// TwinCAT 3 PLC project myPLC
// ProgramVersion: 3.1.4026.21
// CompilerDefines: VISU_USEPROPERTYINFO
// libraries:
//   CmpBitmapPool, * (System)
//   Tc2_Standard, * (Beckhoff Automation GmbH)
//   Tc2_System, * (Beckhoff Automation GmbH)
// project tree:
//   DUTs/ sysInputs.TcDUT, sysOutputs.TcDUT, sysRpiWatchdog.TcDUT, sysState.TcDUT, sysTimersCounters.TcDUT, sysTransitions.TcDUT, sysType.TcDUT
//   / GlobalTextList.TcGTLO, ImagePool.TcIPO (not stored), PlcTask.TcTTO, PlcTask_1.TcTTO, TextList.TcTLO, Visualization Manager.TcVMO (not stored)
//   GVLs/ alarm_global.TcGVL
//   POUs/ FB_EMERGENCY_SYS.TcPOU, FB_HMI_CTRL.TcPOU, FB_RPi_WATCHDOG.TcPOU, FB_STEPPER_CTRL.TcPOU, MAIN.TcPOU, PWM.TcPOU
//   VISUs/ HMI.TcVIS, Visualization.TcVIS
// real-time tasks:
//   TASK PlcTask: cycle T#10ms, priority 20, ADS port 350
//   TASK PWM: cycle T#1ms, priority 1, ADS port 351
//   TASK VISU_TASK: cycle T#200000us, priority 30, ADS port 352
// I/O:
//   DEVICE Device 2 (EtherCAT), AmsNetId 5.144.153.185.3.1
//     Term 1 (EK1100) [EK1100 EtherCAT Coupler (2A E-Bus)]
//       Term 2 (EL5101) [EL5101 1Ch. Inc. Encoder 5V]
//       Term 3 (EL2008) [EL2008 8Ch. Dig. Output 24V, 0.5A]
//       Term 4 (EL4031) [EL4031 1Ch. Ana. Output +/-10V, 12bit]
//       Term 5 (EL1008) [EL1008 8Ch. Dig. Input 24V, 3ms]
//       Term 6 (EL9011) [EL9011 End Terminal]
// variable links:
//   myPLC/myPLC Instance <-> Device 2 (EtherCAT)/Term 1 (EK1100)/Term 3 (EL2008)
//     PlcTask Outputs/PWM.bAlarmaOut <-> Channel 6/Output
//     PlcTask_1 Outputs/MAIN.stSystem.outputs.oMotorDir <-> Channel 7/Output
//     PlcTask_1 Outputs/MAIN.stSystem.outputs.oMotorPulse <-> Channel 8/Output
//   myPLC/myPLC Instance <-> Device 2 (EtherCAT)/Term 1 (EK1100)/Term 5 (EL1008)
//     PlcTask_1 Inputs/MAIN.stSystem.inputs.iAlarmButton_preFtrig_physical <-> Channel 7/Input
//     PlcTask_1 Inputs/MAIN.stSystem.inputs.iSwitch_physical <-> Channel 3/Input
//     PlcTask_1 Inputs/MAIN.stSystem.inputs.iTestButton_preRtrig_physical <-> Channel 5/Input
//     PlcTask_1 Inputs/MAIN.stSystem.inputs.ilimitSwitchClose_preRtrig <-> Channel 8/Input
//     PlcTask_1 Inputs/MAIN.stSystem.inputs.ilimitSwitchOpen_preRtrig <-> Channel 4/Input

CONFIGURATION myPLC
    RESOURCE PLC ON TwinCAT3
        TASK PlcTask(INTERVAL := T#1ms, PRIORITY := 1);
        TASK PlcTask_1(INTERVAL := T#10ms, PRIORITY := 20);
        PROGRAM PWM WITH PlcTask : PWM;
        PROGRAM MAIN WITH PlcTask_1 : MAIN;
    END_RESOURCE
END_CONFIGURATION

// ---- DUTs/sysInputs.TcDUT
TYPE sysInputs :
STRUCT
	
	
	iSwitch_physical         AT %I*: BOOL;   // antes: iSwitch
	iAlarmButton_preFtrig_physical AT %I*: BOOL;  // antes: iAlarmButton_preFtrig
	iTestButton_preRtrig_physical  AT %I*: BOOL;  // antes: iTestButton_preRtrig

	
	iFacialDetec AT %I*: BOOL;
	
	iAlarmButton_ftrig : F_TRIG;
	iTestButton_rtrig	 : R_TRIG;
	
	iAlarmButton : BOOL;
	iTestbutton: BOOL;
	
	
	iHoldAlarm : BOOL;
	iHoldTest : BOOL;
	iHoldAlarm_HMI: BOOL;
	iHoldTest_HMI : BOOL;
	

	
	limitSwitchOpen_rtrig : F_TRIG;
	limitSwitchClose_rtrig : R_TRIG;
	
	ilimitSwitchOpen : BOOL;
	ilimitSwitchClose: BOOL;
	
	ilimitSwitchOpen_preRtrig AT %I* : BOOL;
	ilimitSwitchClose_preRtrig AT %I* : BOOL;
	
	//HMI VARIABLES
	iSwitch_HMI          : BOOL;
    iAlarmButton_HMI     : BOOL;
    iTestButton_HMI      : BOOL;
	iSwitch              : BOOL;
	iAlarmButton_preFtrig: BOOL;
	iTestButton_preRtrig : BOOL;

	
END_STRUCT
END_TYPE

// ---- DUTs/sysOutputs.TcDUT
TYPE sysOutputs :
STRUCT
	
	oAlarm		AT %Q*: BOOL;
	oCloseDoor	AT %Q*: BOOL;
	oOpenDoor	AT %Q*: BOOL;
	
	// MOTOR NEMA17 / TB6600
    oMotorPulse AT %Q*: BOOL;   // → PUL- del TB6600
    oMotorDir   AT %Q*: BOOL;   // → DIR- del TB6600

	//
	oLightGreen  : BOOL;
	oLightOrange : BOOL;
	oLightRed    : BOOL;

	
END_STRUCT
END_TYPE

// ---- DUTs/sysRpiWatchdog.TcDUT
TYPE sysRpiWatchdog :
STRUCT

	iHeartbeat      : INT; // RECEIVED VALUE
	iHeartbeatEcho	: INT;  // VALUE TO SEND
	
	iRPiFail	 AT %I*: BOOL	:= FALSE;


END_STRUCT
END_TYPE

// ---- DUTs/sysState.TcDUT
{attribute 'qualified_only'}
{attribute 'strict'}
{attribute 'to_string'}
TYPE sysState :
(
    stDisconnected := 0,
    stOpening := 1,
    stClosing := 2,
    stWaitingRaspberry := 3,
    stAlarmOpening := 4,
    stAlarm := 5,
    stAlarmClosing := 6,
    stFaceDetectionAlarmOpening := 7,
    stFaceDetectionAlarm := 8,
    stFaceDetectionAlarmClosing := 9,
    stConfigOpening := 10,
    stConfig := 11,
    stConfigClosing := 12,
    stRaspberryFailOpening := 13,
    stRaspberryFail := 14
);
END_TYPE

// ---- DUTs/sysTimersCounters.TcDUT
TYPE sysTimersCounters :
STRUCT
	
	doorOpenTimer : TON;
	doorCloseTimer : TON;
	rpiPingTimer : TON;
	rpiWaitTimer : TON;


	testButtonTimer : TON;
	alarmButtonTImer : TON; 
	alarmButtonTimer_HMI : TON;
	testButtonTimer_HMI  : TON;

	
	
END_STRUCT

END_TYPE

// ---- DUTs/sysTransitions.TcDUT
TYPE sysTransitions :
STRUCT
    T1 : BOOL;
    T2 : BOOL;
    T3 : BOOL;
    T4 : BOOL;
    T5 : BOOL;
    T6 : BOOL;
    T7 : BOOL;
    T8 : BOOL;
    T9 : BOOL;
    T10 : BOOL;
    T11 : BOOL;
    T12 : BOOL;
    T13 : BOOL;
    T14 : BOOL;
    T15 : BOOL;
    T16 : BOOL;
    T17 : BOOL;
    T18 : BOOL;
    T19 : BOOL;
    T20 : BOOL;
    T21 : BOOL;
    T22 : BOOL;
    T23 : BOOL;
    T24 : BOOL;
    T25 : BOOL;
    T26 : BOOL;
    T27 : BOOL;
    T28 : BOOL;
    T29 : BOOL;
    T30 : BOOL;
    T31 : BOOL;
    T32 : BOOL;
    T33 : BOOL;
    T34 : BOOL;
    T35 : BOOL;
    T36 : BOOL;
    T37 : BOOL;

END_STRUCT
END_TYPE

// ---- DUTs/sysType.TcDUT
TYPE sysType :
STRUCT
	state: sysState ;
	
	timersCounters: sysTimersCounters;

	transitions: sysTransitions;
	
	inputs: sysInputs;
	outputs: sysOutputs;
	
	RPiWatchdog: sysRpiWatchdog;
	
END_STRUCT
END_TYPE

// ---- GVLs/alarm_global.TcGVL
{attribute 'qualified_only'}
VAR_GLOBAL
	activate_alarm_global : BOOL;
END_VAR

// ---- POUs/PWM.TcPOU
PROGRAM PWM
VAR
    fbTimer : TON;
    bAlarmaOut AT %Q* : BOOL;  // EL2008 ports
    
    rVolume : REAL := 0.0;   // "Volume" (Duty Cycle) from 0.0 to 100.0 %
    tPeriod : TIME := T#50MS; // PWM frequency (20ms = 50Hz)
    tTiempoAlto : TIME;

END_VAR

IF alarm_global.activate_alarm_global THEN
	rVolume := 0.001;
ELSE
	rVolume := 0;
END_IF

// 1. On time calculation
tTiempoAlto := REAL_TO_TIME((rVolume / 100.0) * TIME_TO_REAL(tPeriod));

// 2. Timer that resets each cycle
fbTimer(IN:= NOT fbTimer.Q, PT:= tPeriod);

// 3. PWM Logic
IF rVolume <= 0.0 THEN
    bAlarmaOut := FALSE; // Power off
ELSIF rVolume >= 100.0 THEN
    bAlarmaOut := TRUE;  // Porwen on
ELSE
    // Elapsed time < up_time -> power on, else power off
    bAlarmaOut := (fbTimer.ET <= tTiempoAlto);
END_IF

END_PROGRAM

// ---- POUs/MAIN.TcPOU
// /////////////////////////////////////////////////////////////////////////////
// ///                                                                       ///
// ///    SYSTEM:     AIRPORT EMERGENCY DOOR                                 ///
// ///                                                                       ///
// ///                                                                       ///
// ///    SUBJECT:       AUTOMATION AND INDUSTRIAL INSTRUMENTATION           ///
// ///    DATE:       2026-04-01                                             ///
// ///                                                                       ///
// ///    MADE BY:    [01] Iñigo Bañuls                                      ///
// ///                [02] Lander Nieto                                      ///
// ///                [03] Ruud Rohan                                        ///
// ///                                                                       ///
// /////////////////////////////////////////////////////////////////////////////



PROGRAM MAIN
VAR
	{attribute 'OPC.UA.DA' := '1'}
	stSystem	:	sysType;                  // SYSTEM DATA STRUCT
	EMERGENCY_HDL	: FB_EMERGENCY_SYS;		  // EMERGENCY HANDLING FUNCTION BLOCK	
	RPi_WATCHDOG	: FB_RPi_WATCHDOG;
	
	
	HMI_CTRL      : FB_HMI_CTRL;

	
	
	STEPPER_CTRL    : FB_STEPPER_CTRL;		  // STEPPER MOTOR CONTROL
    bIsOpening      : BOOL;
    bIsClosing      : BOOL;
	
	
	
// Atributos para exponer las variables al servidor OPC UA
    {attribute 'OPC.UA.DA' := '1'}
    aImageRxBuffer : ARRAY[0..99999] OF BYTE; // Buffer para recibir desde la RPi (Ej: 100 KB)
    
    {attribute 'OPC.UA.DA' := '1'}
    aImageTxBuffer : ARRAY[0..99999] OF BYTE; // Buffer para enviar a la RPi
    
    // Variables de control (Handshake)
    {attribute 'OPC.UA.DA' := '1'}
    bRpiHasWritten : BOOL; // La RPi lo pone en TRUE cuando termina de enviar
    
    {attribute 'OPC.UA.DA' := '1'}
    bPlcHasWritten : BOOL; // El PLC lo pone en TRUE cuando tiene una imagen lista para la RPi

	
END_VAR

EMERGENCY_HDL(stSystem := stSystem);
RPi_WATCHDOG(stSystem := stSystem);
EMERGENCY_HDL.mTransitions(stSystem := stSystem);
EMERGENCY_HDL.mOutputs(stSystem := stSystem);
HMI_CTRL(stSystem := stSystem);

STEPPER_CTRL(
    bOpen   := stSystem.outputs.oOpenDoor,
    bClose  := stSystem.outputs.oCloseDoor,
    bEnable := NOT (stSystem.state = sysState.stDisconnected), 
    bPulse  => stSystem.outputs.oMotorPulse,
    bDir    => stSystem.outputs.oMotorDir
);

END_PROGRAM

// ---- POUs/FB_EMERGENCY_SYS.TcPOU
FUNCTION_BLOCK FB_EMERGENCY_SYS
VAR_IN_OUT
	stSystem: sysType;         // ALLOW CHILD METHODS TO ACCESS DATA
END_VAR

CASE stSystem.state OF

    // ==========================================
    // INITIAL STATES
    // ==========================================
    sysState.stDisconnected:
        IF stSystem.transitions.T1 THEN
            stSystem.state := sysState.stClosing;
        END_IF

    sysState.stOpening:
        IF stSystem.transitions.T2 THEN
            stSystem.state := sysState.stDisconnected;
        END_IF

    sysState.stClosing:
        IF stSystem.transitions.T3 THEN
            stSystem.state := sysState.stWaitingRaspberry;
        END_IF

    // ==========================================
    // WAIT AND RASPBERRY CONNECTION
    // ==========================================
    sysState.stWaitingRaspberry:
        IF stSystem.transitions.T4 THEN
            stSystem.state := sysState.stOpening;
        ELSIF stSystem.transitions.T7 THEN
            stSystem.state := sysState.stAlarmOpening;
        ELSIF stSystem.transitions.T8 THEN
            stSystem.state := sysState.stFaceDetectionAlarmOpening;
        ELSIF stSystem.transitions.T9 THEN
            stSystem.state := sysState.stConfigOpening;
        ELSIF stSystem.transitions.T5 THEN
            stSystem.state := sysState.stRaspberryFailOpening;
        END_IF


    // ==========================================
    // DEFAULT ALARM
    // ==========================================
    sysState.stAlarmOpening:
        IF stSystem.transitions.T15 THEN
            stSystem.state := sysState.stAlarm;
        ELSIF stSystem.transitions.T37 THEN
            stSystem.state := sysState.stAlarmClosing;
        END_IF

    sysState.stAlarm:
        IF stSystem.transitions.T16 THEN
            stSystem.state := sysState.stAlarmClosing;
        END_IF

    sysState.stAlarmClosing:
        IF stSystem.transitions.T17 THEN
            stSystem.state := sysState.stWaitingRaspberry;
        ELSIF stSystem.transitions.T26 THEN
            stSystem.state := sysState.stAlarmOpening;
        ELSIF stSystem.transitions.T27 THEN
            stSystem.state := sysState.stFaceDetectionAlarmOpening;
        ELSIF stSystem.transitions.T28 THEN
            stSystem.state := sysState.stConfigOpening;
        END_IF

    // ==========================================
    // FACIAL DETECTION ALARM
    // ==========================================
    sysState.stFaceDetectionAlarmOpening:
        IF stSystem.transitions.T18 THEN
            stSystem.state := sysState.stFaceDetectionAlarm;
        ELSIF stSystem.transitions.T35 THEN
            stSystem.state := sysState.stFaceDetectionAlarmClosing;
        END_IF

    sysState.stFaceDetectionAlarm:
        IF stSystem.transitions.T19 THEN
            stSystem.state := sysState.stFaceDetectionAlarmClosing;
        END_IF

    sysState.stFaceDetectionAlarmClosing:
        IF stSystem.transitions.T20 THEN
            stSystem.state := sysState.stWaitingRaspberry;
        ELSIF stSystem.transitions.T29 THEN
            stSystem.state := sysState.stAlarmOpening;
        ELSIF stSystem.transitions.T30 THEN
            stSystem.state := sysState.stFaceDetectionAlarmOpening;
        ELSIF stSystem.transitions.T31 THEN
            stSystem.state := sysState.stConfigOpening;
        END_IF

    // ==========================================
    // TEST MODE
    // ==========================================
    sysState.stConfigOpening:
        IF stSystem.transitions.T21 THEN
            stSystem.state := sysState.stConfig;
        ELSIF stSystem.transitions.T36 THEN
            stSystem.state := sysState.stConfigClosing;
        END_IF

    sysState.stConfig:
        IF stSystem.transitions.T22 THEN
            stSystem.state := sysState.stConfigClosing;
        END_IF

    sysState.stConfigClosing:
        IF stSystem.transitions.T23 THEN
            stSystem.state := sysState.stWaitingRaspberry;
        ELSIF stSystem.transitions.T32 THEN
            stSystem.state := sysState.stAlarmOpening;
        ELSIF stSystem.transitions.T33 THEN
            stSystem.state := sysState.stFaceDetectionAlarmOpening;
        ELSIF stSystem.transitions.T34 THEN
            stSystem.state := sysState.stConfigOpening;
        END_IF

    // ==========================================
    // RASPBERRY PI ERROR
    // ==========================================
    sysState.stRaspberryFailOpening:
        IF stSystem.transitions.T24 THEN
            stSystem.state := sysState.stRaspberryFail;
        END_IF

    sysState.stRaspberryFail:
        IF stSystem.transitions.T25 THEN
            stSystem.state := sysState.stDisconnected;
        END_IF

END_CASE

METHOD mOutputs
VAR_IN_OUT
    stSystem: sysType;
END_VAR
// ==============================================================================
// Method: mOutputs
// Description: Triggers corresponding outputs in each state
// ==============================================================================

stSystem.outputs.oOpenDoor :=
    (stSystem.state = sysState.stOpening) OR
    (stSystem.state = sysState.stAlarmOpening) OR
    (stSystem.state = sysState.stFaceDetectionAlarmOpening) OR
    (stSystem.state = sysState.stConfigOpening) OR
    (stSystem.state = sysState.stRaspberryFailOpening);

// --- oCloseDoor: active in all Closing states ---
stSystem.outputs.oCloseDoor :=
    (stSystem.state = sysState.stClosing) OR
    (stSystem.state = sysState.stAlarmClosing) OR
    (stSystem.state = sysState.stFaceDetectionAlarmClosing) OR
    (stSystem.state = sysState.stConfigClosing);

// --- oAlarm: active during any alarm state (both alarm types, all sub-states) ---
alarm_global.activate_alarm_global :=
    (stSystem.state = sysState.stAlarmOpening) OR
    (stSystem.state = sysState.stAlarm) OR
    (stSystem.state = sysState.stAlarmClosing) OR
    (stSystem.state = sysState.stFaceDetectionAlarmOpening) OR
    (stSystem.state = sysState.stFaceDetectionAlarm) OR
    (stSystem.state = sysState.stFaceDetectionAlarmClosing) OR
(stSystem.state = sysState.stRaspberryFailOpening) OR
(stSystem.state = sysState.stRaspberryFail);


// Green: door is opened
stSystem.outputs.oLightGreen :=
    (stSystem.state = sysState.stAlarm) OR
    (stSystem.state = sysState.stFaceDetectionAlarm) OR
    (stSystem.state = sysState.stConfig) OR
    (stSystem.state = sysState.stRaspberryFail) OR
    (stSystem.state = sysState.stDisconnected);

// Yellow: door is moving
stSystem.outputs.oLightOrange :=
    (stSystem.state = sysState.stOpening) OR
    (stSystem.state = sysState.stClosing) OR
    (stSystem.state = sysState.stAlarmOpening) OR
    (stSystem.state = sysState.stAlarmClosing) OR
    (stSystem.state = sysState.stFaceDetectionAlarmOpening) OR
    (stSystem.state = sysState.stFaceDetectionAlarmClosing) OR
    (stSystem.state = sysState.stConfigOpening) OR
    (stSystem.state = sysState.stConfigClosing) OR
    (stSystem.state = sysState.stRaspberryFailOpening);

// Red: door is closed
stSystem.outputs.oLightRed :=
    (stSystem.state = sysState.stWaitingRaspberry);
END_METHOD

METHOD mTransitions : BOOL
VAR_IN_OUT
    stSystem: sysType;
	
	
END_VAR
// ==============================================================================
// Method: mTransitions
// Description: Evaluates and triggers the boolean flags for state transitions
//              based on the current state and specific logical conditions.
// ==============================================================================

stSystem.inputs.iSwitch := stSystem.inputs.iSwitch_physical OR stSystem.inputs.iSwitch_HMI;

stSystem.inputs.iAlarmButton_preFtrig := stSystem.inputs.iAlarmButton_preFtrig_physical;
stSystem.inputs.iTestButton_preRtrig  := stSystem.inputs.iTestButton_preRtrig_physical;

	
stSystem.inputs.limitSwitchClose_rtrig(CLK := stSystem.inputs.ilimitSwitchClose_preRtrig, Q => stSystem.inputs.ilimitSwitchClose);
stSystem.inputs.limitSwitchOpen_rtrig(CLK := stSystem.inputs.ilimitSwitchOpen_preRtrig, Q => stSystem.inputs.ilimitSwitchOpen);

stSystem.inputs.iAlarmButton_ftrig(CLK:= stSystem.inputs.iAlarmButton_preFtrig,Q => stSystem.inputs.iAlarmButton);
stSystem.inputs.iTestButton_rtrig(CLK:= stSystem.inputs.iTestButton_preRtrig, Q => stSystem.inputs.iTestbutton);

stSystem.timersCounters.alarmButtonTImer(
	 IN := NOT stSystem.inputs.iAlarmButton_preFtrig,
	 PT := T#5S,
	 Q => stSystem.inputs.iHoldAlarm
);
stSystem.timersCounters.testButtonTimer(
	IN := stSystem.inputs.iTestButton_preRtrig, 
	PT := T#5S, 
	Q => stSystem.inputs.iHoldTest
);

stSystem.timersCounters.alarmButtonTimer_HMI(
    IN := stSystem.inputs.iAlarmButton_HMI,
    PT := T#5S,
    Q => stSystem.inputs.iHoldAlarm_HMI
);
stSystem.timersCounters.testButtonTimer_HMI(
    IN := stSystem.inputs.iTestButton_HMI,
    PT := T#5S,
    Q => stSystem.inputs.iHoldTest_HMI
);

// Transition T1: FROM stDisconnected TO stClosing WHEN iSwitch is TRUE
stSystem.transitions.T1 := (stSystem.state = sysState.stDisconnected) AND (stSystem.inputs.iSwitch = TRUE);

// Transition T2: FROM stOpening TO stDisconnected WHEN doorOpenTimer is done
stSystem.transitions.T2 := (stSystem.state = sysState.stOpening) AND (stSystem.inputs.ilimitSwitchOpen = TRUE);

// Transition T3: FROM stClosing TO stWaitingRaspberry WHEN doorCloseTimer is done
stSystem.transitions.T3 := (stSystem.state = sysState.stClosing) AND (stSystem.inputs.ilimitSwitchClose = TRUE);

// Transition T4: FROM stWaitingRaspberry TO stOpening WHEN iSwitch is FALSE
stSystem.transitions.T4 := (stSystem.state = sysState.stWaitingRaspberry) AND (stSystem.inputs.iSwitch = FALSE);

// ... you must continue this pattern up to T25 following the transition table.

// T5: FROM stWaitingRaspberry TO stRaspberryFailOpening WHEN iRPiFail TRUE
stSystem.transitions.T5 := (stSystem.state = sysState.stWaitingRaspberry) AND (stSystem.RPiWatchdog.iRPiFail = TRUE);


// T7: FROM stWaitingRaspberry TO stAlarmOpening WHEN alarm button pressed
stSystem.transitions.T7 := (stSystem.state = sysState.stWaitingRaspberry) 
    AND (stSystem.inputs.iHoldAlarm = TRUE OR stSystem.inputs.iHoldAlarm_HMI = TRUE);

// T8: FROM stWaitingRaspberry TO stFaceDetectionAlarmOpening WHEN face detected
stSystem.transitions.T8 := (stSystem.state = sysState.stWaitingRaspberry) AND (stSystem.inputs.iFacialDetec = TRUE);
 	
// T9: FROM stWaitingRaspberry TO stConfigOpening WHEN test button pressed
stSystem.transitions.T9 := (stSystem.state = sysState.stWaitingRaspberry) 
    AND (stSystem.inputs.iHoldTest = TRUE OR stSystem.inputs.iHoldTest_HMI = TRUE);

// T15: FROM stAlarmOpening TO stAlarm WHEN doorOpenTimer done
stSystem.transitions.T15 := (stSystem.state = sysState.stAlarmOpening) AND (stSystem.inputs.ilimitSwitchOpen = TRUE);

// T16: FROM stAlarm TO stAlarmClosing WHEN test button AND alarm cleared
stSystem.transitions.T16 := (stSystem.state = sysState.stAlarm) 
    AND (stSystem.inputs.iTestButton_preRtrig = TRUE OR stSystem.inputs.iTestButton_HMI = TRUE)
    AND (stSystem.inputs.iAlarmButton_preFtrig = TRUE OR stSystem.inputs.iAlarmButton_HMI = TRUE);


// T17: FROM stAlarmClosing TO stWaitingRaspberry WHEN doorCloseTimer done
stSystem.transitions.T17 := (stSystem.state = sysState.stAlarmClosing) AND (stSystem.inputs.ilimitSwitchClose = TRUE);

// T18: FROM stFaceDetectionAlarmOpening TO stFaceDetectionAlarm WHEN doorOpenTimer done
stSystem.transitions.T18 := (stSystem.state = sysState.stFaceDetectionAlarmOpening) AND (stSystem.inputs.ilimitSwitchOpen = TRUE);

// T19: FROM stFaceDetectionAlarm TO stFaceDetectionAlarmClosing WHEN test button AND alarm cleared
stSystem.transitions.T19 := (stSystem.state = sysState.stFaceDetectionAlarm) 
    AND (stSystem.inputs.iTestButton = TRUE OR stSystem.inputs.iTestButton_HMI = TRUE)
    AND (stSystem.inputs.iAlarmButton = TRUE OR stSystem.inputs.iAlarmButton_HMI = TRUE);

// T20: FROM stFaceDetectionAlarmClosing TO stWaitingRaspberry WHEN doorCloseTimer done
stSystem.transitions.T20 := (stSystem.state = sysState.stFaceDetectionAlarmClosing) AND (stSystem.inputs.ilimitSwitchClose = TRUE);

// T21: FROM stConfigOpening TO stConfig WHEN doorOpenTimer done
stSystem.transitions.T21 := (stSystem.state = sysState.stConfigOpening) AND (stSystem.inputs.ilimitSwitchOpen = TRUE);

// T22: FROM stConfig TO stConfigClosing WHEN test button pressed
stSystem.transitions.T22 := (stSystem.state = sysState.stConfig) AND (stSystem.inputs.iTestButton = TRUE);

// T23: FROM stConfigClosing TO stWaitingRaspberry WHEN doorCloseTimer done
stSystem.transitions.T23 := (stSystem.state = sysState.stConfigClosing) AND (stSystem.inputs.ilimitSwitchClose= TRUE);

// T24: FROM stRaspberryFailOpening TO stRaspberryFail WHEN doorOpenTimer done
stSystem.transitions.T24 := (stSystem.state = sysState.stRaspberryFailOpening) AND (stSystem.inputs.ilimitSwitchOpen = TRUE);

// T25: FROM stRaspberryFail TO stDisconnected WHEN iSwitch is FALSE
stSystem.transitions.T25 := (stSystem.state = sysState.stRaspberryFail) AND (stSystem.inputs.iSwitch = FALSE);

// T26: FROM stAlarmClosing TO stAlarmOpening WHEN alarm button pressed
stSystem.transitions.T26 := (stSystem.state = sysState.stAlarmClosing) AND (stSystem.inputs.iHoldAlarm = TRUE);

// T27: FROM stAlarmClosing TO stFaceDetectionAlarmOpening WHEN face detected
stSystem.transitions.T27 := (stSystem.state = sysState.stAlarmClosing) AND (stSystem.inputs.iFacialDetec = TRUE);

// T28: FROM stAlarmClosing TO stConfigOpening WHEN test button pressed
stSystem.transitions.T28 := (stSystem.state = sysState.stAlarmClosing) AND (stSystem.inputs.iHoldTest = TRUE);

// T29: FROM stFaceDetectionAlarmClosing TO stAlarmOpening WHEN alarm button pressed
stSystem.transitions.T29 := (stSystem.state = sysState.stFaceDetectionAlarmClosing) AND (stSystem.inputs.iHoldAlarm = TRUE);

// T30: FROM stFaceDetectionAlarmClosing TO stFaceDetectionAlarmOpening WHEN face detected
stSystem.transitions.T30 := (stSystem.state = sysState.stFaceDetectionAlarmClosing) AND (stSystem.inputs.iFacialDetec = TRUE);

// T31: FROM stFaceDetectionAlarmClosing TO stConfigOpening WHEN test button pressed
stSystem.transitions.T31 := (stSystem.state = sysState.stFaceDetectionAlarmClosing) AND (stSystem.inputs.iHoldTest = TRUE);

// T32: FROM stConfigClosing TO stAlarmOpening WHEN alarm button pressed
stSystem.transitions.T32 := (stSystem.state = sysState.stConfigClosing) AND (stSystem.inputs.iHoldAlarm = TRUE);

// T33: FROM stConfigClosing TO stFaceDetectionAlarmOpening WHEN face detected
stSystem.transitions.T33 := (stSystem.state = sysState.stConfigClosing) AND (stSystem.inputs.iFacialDetec = TRUE);

// T34: FROM stConfigClosing TO stConfigOpening WHEN test button pressed
stSystem.transitions.T34 := (stSystem.state = sysState.stConfigClosing) AND (stSystem.inputs.iHoldTest = TRUE);

// T35: FROM stFaceDetectionAlarmOpening TO stFaceDetectionAlarmClosing WHEN test button AND alarm cleared
stSystem.transitions.T35 := (stSystem.state = sysState.stFaceDetectionAlarmOpening) 
    AND (stSystem.inputs.iTestButton = TRUE OR stSystem.inputs.iTestButton_HMI = TRUE)
    AND (stSystem.inputs.iAlarmButton = TRUE OR stSystem.inputs.iAlarmButton_HMI = TRUE);


// T36: FROM stConfigOpening TO stConfigClosing WHEN test button AND alarm cleared
stSystem.transitions.T36 := (stSystem.state = sysState.stConfigOpening) 
    AND (stSystem.inputs.iTestButton = TRUE OR stSystem.inputs.iTestButton_HMI = TRUE)
    AND (stSystem.inputs.iAlarmButton = TRUE OR stSystem.inputs.iAlarmButton_HMI = TRUE);


// T37: FROM stAlarmOpening TO stAlarmClosing WHEN test button AND alarm cleared
stSystem.transitions.T37 := (stSystem.state = sysState.stAlarmOpening) 
    AND (stSystem.inputs.iTestButton = TRUE OR stSystem.inputs.iTestButton_HMI = TRUE)
    AND (stSystem.inputs.iAlarmButton = TRUE OR stSystem.inputs.iAlarmButton_HMI = TRUE);
END_METHOD

END_FUNCTION_BLOCK

// ---- POUs/FB_RPi_WATCHDOG.TcPOU
FUNCTION_BLOCK FB_RPi_WATCHDOG
VAR
    //iHeartbeat      : INT; // RECEIVED VALUE
    iHeartbeat_Prev : INT; // PREV VALUE REGISTRY
    
    fbWatchdog      : TON; // WATCHDOG TIMER
    bRaspberryFail  : BOOL; // ERROR FLAG TO BE SUBSTITUDED
	
	//iHeartbeatEcho	: INT;  // VALUE TO SEND
END_VAR

VAR_IN_OUT
	stSystem: sysType;       
END_VAR

// 1. Timer Init
// If new received value equals value received before, no new value was received
// This controls IN port. While the values are equal, it counts.
fbWatchdog(IN := (stSystem.RPiWatchdog.iHeartbeat = iHeartbeat_Prev), PT := T#3S); 


// If timer runs out
IF fbWatchdog.Q THEN
    bRaspberryFail := TRUE; 
	
ELSE
    bRaspberryFail := FALSE;
END_IF

// 3. Echo and mem update
stSystem.RPiWatchdog.iHeartbeatEcho := stSystem.RPiWatchdog.iHeartbeat;       // Echoes the message to the RPi
iHeartbeat_Prev := stSystem.RPiWatchdog.iHeartbeat;       // Value is logged
stSystem.RPiWatchdog.iRPiFail := bRaspberryFail;

END_FUNCTION_BLOCK

// ---- POUs/FB_HMI_CTRL.TcPOU
FUNCTION_BLOCK FB_HMI_CTRL
VAR_IN_OUT
    stSystem : sysType; 
END_VAR
VAR_OUTPUT
    sImagenActual : STRING; // Image ID
END_VAR

CASE stSystem.state OF
    
    // default
    sysState.stDisconnected, sysState.stClosing, sysState.stOpening:
        sImagenActual := 'opened';

    // alarm
    sysState.stWaitingRaspberry:
        sImagenActual := 'closed';

    // facial alamar
    sysState.stFaceDetectionAlarmOpening, sysState.stFaceDetectionAlarm, sysState.stFaceDetectionAlarmClosing:
        sImagenActual := 'terrorist';

    // configuration state
    sysState.stConfigOpening, sysState.stConfig, sysState.stConfigClosing:
        sImagenActual := 'config';
		
	// hacked state
    sysState.stRaspberryFailOpening, sysState.stRaspberryFail:
        sImagenActual := 'hackeado';


    sysState.stAlarmOpening, sysState.stAlarm, sysState.stAlarmClosing :
        sImagenActual := 'alarm';

ELSE
    sImagenActual := '';
END_CASE

END_FUNCTION_BLOCK

// ---- POUs/FB_STEPPER_CTRL.TcPOU
FUNCTION_BLOCK FB_STEPPER_CTRL
VAR_INPUT
    bOpen   : BOOL;
    bClose  : BOOL;
    bEnable : BOOL;
END_VAR
VAR_OUTPUT
    bPulse  : BOOL;
    bDir    : BOOL;
END_VAR
VAR
    tonON   : TON;
    tonOFF  : TON;
END_VAR

IF bEnable AND (bOpen OR bClose) THEN

    // Timer ON: wait 10 ms, then pulse
    tonON(IN := NOT bPulse, PT := T#1MS);
    IF tonON.Q THEN
        bPulse := TRUE;
    END_IF

    // Timer OFF: when pulse is ready, wait 10 ms and quit
    tonOFF(IN := bPulse, PT := T#1MS);
    IF tonOFF.Q THEN
        bPulse := FALSE;
    END_IF

    // Direction, depending on what is activated
    bDir := bOpen;

ELSE
    // Reset when motor is stopped
    bPulse := FALSE;
    bDir   := FALSE;
    tonON(IN := FALSE);
    tonOFF(IN := FALSE);
END_IF

END_FUNCTION_BLOCK

// ---- GlobalTextList.TcGTLO
TEXTLIST GlobalTextList
  95 = '%s'
  668 = 'CASTELL'
  364 = 'CASTELLANO'
  223 = 'ENGLISH'
END_TEXTLIST

// ---- TextList.TcTLO
TEXTLIST TextList
  1 = 'ESTADO DE LA ALARMA'
  2 = 'ABIERTO' | English: 'OPENED' | Spanish: 'ABIERTO'
  3 = 'ABRIENDO/\nCERRANDO' | English: 'OPENING/\nCLOSING' | Spanish: 'ABRIENDO/\nCERRANDO'
  4 = 'CERRADO' | English: 'CLOSED' | Spanish: 'CERRADO'
  5 = 'INTERRUPTOR' | English: 'SWITCH' | Spanish: 'INTERRUPTOR'
  6 = 'ALARMA' | English: 'ALARM' | Spanish: 'ALARMA'
  7 = 'CONFIGURACIÓN' | English: 'CONFIGURATION' | Spanish: 'CONFIGURACIÓN'
  0 = 'CONECTAR\n/DESCONECTAR \nPUERTA EMERGENCIA' | English: 'CONNECT/\nDISCONNECT\n EMERGENCY DOOR' | Spanish: 'CONECTAR/\nDESCONECTAR \nPUERTA EMERGENCIA'
  9 = 'PUERTA DE EMERGENCIA' | English: 'EMERGENCY DOOR' | Spanish: 'PUERTA DE EMERGENCIA'
   = ''
END_TEXTLIST

// ---- VISUs/HMI.TcVIS
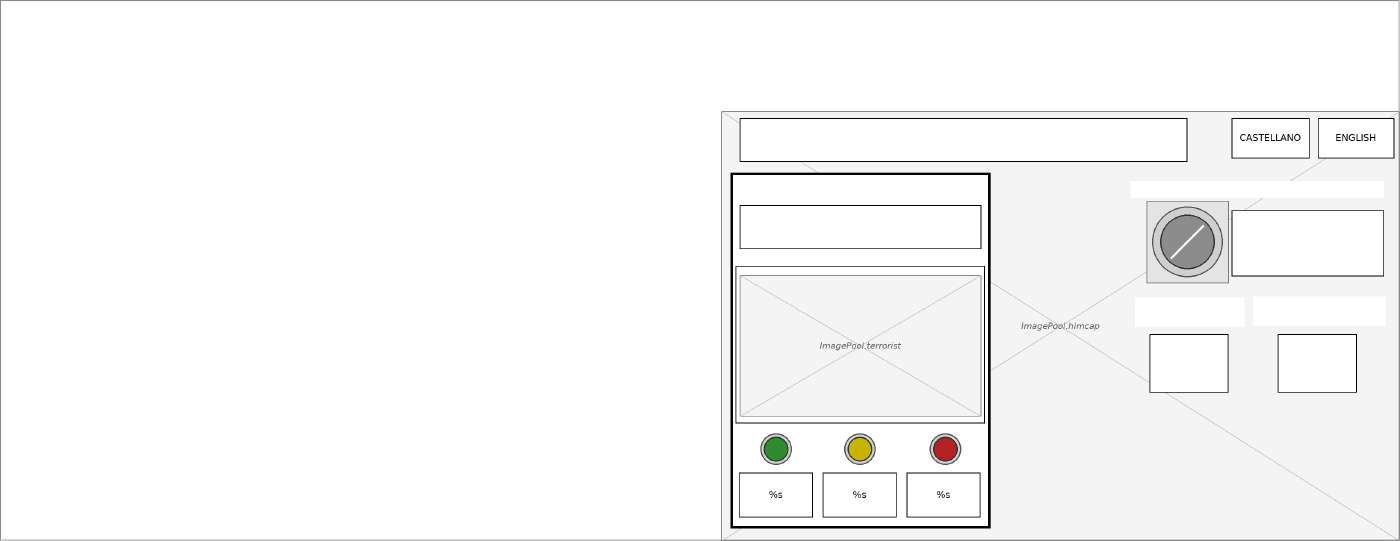
VISUALIZATION HMI  // 1637x633
    Image (843,130 794x503), image: ImagePool.himcap
    RoundedRectangle (854,202 304x416)
    Rectangle (860,311 291x184)
    Image (865,322 282x165), image: ImagePool.terrorist
        p84334746: MAIN.HMI_CTRL.sImagenActual
    RotarySwitch (1339,235 99x96), variable: MAIN.EMERGENCY_HDL.stSystem.inputs.iSwitch_HMI, behaviour: TOGGLE, style: Switch-RotarySwitch-Gray
    RoundedRectangle (1494,391 92x68)
        tap MAIN.EMERGENCY_HDL.stSystem.inputs.iTestButton_HMI
    RoundedRectangle (1344,391 92x68)
        toggle MAIN.EMERGENCY_HDL.stSystem.inputs.iAlarmButton_HMI
    Rectangle (1327,348 128x34), "%s", text list: 'TextList', text index: 6
    Rectangle (1322,212 296x19), "%s", text list: 'TextList', text index: 5
    Lamp1 (886,503 43x45), variable: MAIN.stSystem.outputs.oLightGreen, style: Lamp-Lamp1-Green
    Lamp1 (984,503 43x45), variable: MAIN.stSystem.outputs.oLightOrange, style: Lamp-Lamp1-Yellow
    Lamp1 (1084,503 43x45), variable: MAIN.stSystem.outputs.oLightRed, style: Lamp-Lamp1-Red
    RoundedRectangle (864,553 86x52), "%s", text list: 'TextList', text index: 2
    RoundedRectangle (962,553 86x52), "%s", text list: 'TextList', text index: 3
    RoundedRectangle (1060,553 86x52), "%s", text list: 'TextList', text index: 4
    Rectangle (1465,347 155x34), "%s", text list: 'TextList', text index: 7
    Rectangle (865,240 282x51), "%s", text list: 'TextList', text index: 1
    RoundedRectangle (1541,138 89x47), "ENGLISH"
        OnMouseClick: ChangeLanguage ChangeLanguage=English
    RoundedRectangle (1440,138 91x47), "CASTELLANO"
        OnMouseClick: ChangeLanguage ChangeLanguage=Spanish
    Rectangle (1440,246 178x77), "%s", text list: 'TextList', text index: 0
    Rectangle (865,138 523x51), "%s", text list: 'TextList', text index: 9
END_VISUALIZATION

// ---- VISUs/Visualization.TcVIS
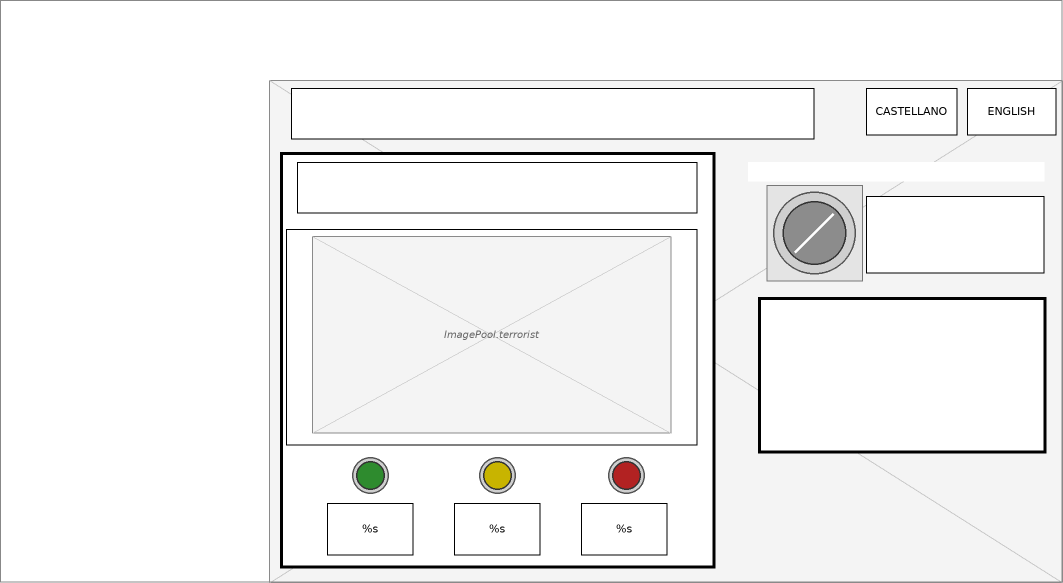
VISUALIZATION Visualization  // 1063x583
    Image (269,80 794x503), image: ImagePool.himcap
    RoundedRectangle (280,152 435x416)
    Rectangle (286,229 411x216)
    Image (312,236 359x197), image: ImagePool.terrorist
        p84334746: MAIN.HMI_CTRL.sImagenActual
    RotarySwitch (765,185 99x96), variable: MAIN.EMERGENCY_HDL.stSystem.inputs.iSwitch_HMI, behaviour: TOGGLE, style: Switch-RotarySwitch-Gray
    Rectangle (748,162 296x19), "%s", text list: 'TextList', text index: 5
    Lamp1 (349,453 43x45), variable: MAIN.stSystem.outputs.oLightGreen, style: Lamp-Lamp1-Green
    Lamp1 (476,453 43x45), variable: MAIN.stSystem.outputs.oLightOrange, style: Lamp-Lamp1-Yellow
    Lamp1 (605,453 43x45), variable: MAIN.stSystem.outputs.oLightRed, style: Lamp-Lamp1-Red
    RoundedRectangle (327,503 86x52), "%s", text list: 'TextList', text index: 2
    RoundedRectangle (454,503 86x52), "%s", text list: 'TextList', text index: 3
    RoundedRectangle (581,503 86x52), "%s", text list: 'TextList', text index: 4
    Rectangle (891,297 155x156)
    Rectangle (297,162 400x51), "%s", text list: 'TextList', text index: 1
    RoundedRectangle (967,88 89x47), "ENGLISH"
        OnMouseClick: ChangeLanguage ChangeLanguage=English
    RoundedRectangle (866,88 91x47), "CASTELLANO"
        OnMouseClick: ChangeLanguage ChangeLanguage=Spanish
    Rectangle (866,196 178x77), "%s", text list: 'TextList', text index: 0
    Rectangle (291,88 523x51), "%s", text list: 'TextList', text index: 9
    RoundedRectangle (758,297 288x156)
        toggle MAIN.EMERGENCY_HDL.stSystem.inputs.iAlarmButton_HMI
    Rectangle (753,360 291x34), "%s", text list: 'TextList', text index: 6
END_VISUALIZATION
